// Mitsubishi GX Works2 project: סופי1   PLC: FX3G

// global labels: Global1
VAR_GLOBAL
  LAMP_WORKDAY AT Y007 : BOOL;  (* נורת חווי יום עבודת פעיל *)
  SW_DAY_START AT X007 : BOOL;  (* מתג תחילת יום *)
  SW_START_PROD AT X001 : BOOL;  (* מתג דגימה של Analog Input *)
  SW_EMERGENCY AT X005 : BOOL;  (* מתג חירום לסיום יום עבודה *)
  LAMP_PREP AT Y000 : BOOL;  (* נורת חווי להכנת הגלידה *)
  SW_COOL AT X002 : BOOL;  (* מתג העברת הגלידות למכלי הקירור *)
  TEMP_SENSOR AT X003 : BOOL;  (* חיישן טמפרטורה *)
  LAMP_COOL AT Y002 : BOOL;  (* נורת חווי לקירור גלידה *)
  LAMP_MIX_A AT Y005 : BOOL;  (* נורת הבהוב לערבוב הגלידה *)
  LAMP_MIX_B AT Y006 : BOOL;  (* נורת הבהוב לערבוב הגלידה *)
  INIT_RASBERRY AT D1700 : REAL;  (* רגיסטר מלאי פטל בתחילת יום *)
  INIT_LEMON AT D1702 : REAL;  (* רגיסטר מלאי לימון בתחילת יום *)
  INIT_STABILIZER AT D1705 : REAL;  (* רגיסטר מלאי מייצב בתחילת יום *)
  INIT_BEARS AT D1111 : REAL;  (* רגיסטר מלאי דובונים בתחילת יום *)
  STOCK_RASBERRY AT D1122 : REAL;  (* רגיסטר מלאי נוכחי פטל *)
  STOCK_LEMON AT D1133 : REAL;  (* רגיסטר מלאי נוכחי לימון *)
  STOCK_STABILIZER AT D1233 : REAL;  (* רגיסטר מלאי נוכחי מייצב *)
  STOCK_BEARS AT D1345 : REAL;  (* רגיסטר מלאי נוכחי דובונים *)
  STORAGE_COUNT AT D2000 : REAL;  (* רגיסטר מיכל מארזים *)
  LAMP_REGULAR AT M1 : BOOL;  (* נורת חיווי עזר להכנת גומיגם רגיל *)
  LAMP_PREMIUM AT M2 : BOOL;  (* נורת חיווי להכנת גומיגם פינוק *)
END_VAR
VAR_GLOBAL CONSTANT
  RESET : REAL;  (* איפוס משתנים *)
  RESET_ANALOG_OUTPUT : INT := K0;  (* איפוס משתנים *)
END_VAR
VAR_GLOBAL
  RAS_COOLING_TANK AT D2100 : REAL;  (* מיכל קירור פטל *)
  LEM_COOLING_TANK AT D2200 : REAL;  (* מיכל קירור לימון *)
END_VAR
VAR_GLOBAL CONSTANT
  RAS_FOR_PREMIUIM : REAL := 385;  (* כמות פטל דרושה למארז פינוק *)
  LEM_FOR_PREMIUIM : REAL := 665;  (* כמות לימון דרושה למארז פינוק *)
  STAB_FOR_PREMIUIM : REAL := 210;  (* כמות חומר מייצב להכנת מארז פינוק *)
  RAS_FOR_CLASSIC : REAL := 280;  (* כמות פטל דרושה למארז רגיל *)
  LEM_FOR_CLASSIC : REAL := 455;  (* כמות לימון דרושה מארז רגיל *)
  STAB_FOR_CLASSIC : REAL := 105;  (* כמות חומר מייצב דרושה מארז רגיל *)
END_VAR
VAR_GLOBAL
  ANALOG_INPUT AT D8280 : INT;  (* משתנה המייצג את סוג המארז *)
  ANALOG_OUTPUT AT D8282 : INT;  (* שעון יציאה אנלוגי למספר מארזים *)
  SAVE_ANALOG_INPUT AT D8201 : INT;  (* משתנה שמירת הדגימה שהתקבלה *)
  LACK_OF_STOCK AT M0 : BOOL;  (* נורת חיווי לסיום יום בשל חוסר בחומרי גלם *)
  INDICATOR_LAMP AT M10 : BOOL;  (* נורת חיווי עזר לבדיקת תקינות ערך אנלוגי *)
END_VAR
VAR_GLOBAL CONSTANT
  MAX_REGULAR : REAL := 5;  (* ערך קלט מקסימום ליצירת מארז רגיל *)
  MIN_PREMIUM : REAL := 6;  (* ערך קלט מקסימום ליצירת מארז פינוק *)
END_VAR
VAR_GLOBAL
  ANALOG_SAMPLED AT D8205 : REAL;  (* רגיסטר של המרת ANALOG_INPUT לFLOAT *)
  CHEKING_FOR_REG AT M3 : BOOL;  (* נורת חווי עזר  לבדיקת מלאי להכנת מארז רגיל *)
  CHECKING_FOR_PREM AT M4 : BOOL;  (* נורת חווי לבדיקת מלאי להכנת מארז פינוק *)
  CONTINUE AT M123 : BOOL;  (* נורת חיווי למעבר להפחתת כמויות ממכלים *)
  ITERATION_LIGHT AT M44 : BOOL;  (* נורת חיווי לסיום איטרציה *)
  START_MIX AT M50 : BOOL;  (* נורת חווי עזר להתחלת ערבוב *)
  MAKING_ICECREAM AT M40 : BOOL;  (* נורת חווי להכנת הגלידה *)
END_VAR
VAR_GLOBAL CONSTANT
  TOTAL_REG_LEM : REAL := 490;  (* כמות גלידה לימון במארז רגיל *)
  TOTAL_PREM_LEM : REAL := 700;  (* כמות גלידה לימון במארז פינוק *)
  TOTAL_REG_RAS : REAL := 350;  (* כמות גלידה פטל במארז רגיל *)
  TOTAL_PREM_RAS : REAL := 560;  (* כמות גלידה פטל במארז פינוק *)
  ICECREAM_MAKING_TIME : INT := 50;  (* משך זמן הכנת גלידה *)
END_VAR
VAR_GLOBAL
  SRART_PACKING AT X006 : BOOL;  (* מתג סיום תהליך ואריזה *)
  PACKING_UNIT AT X000 : BOOL;  (* אריזת יחידה *)
  PACKING_LIGHT AT Y001 : BOOL;  (* נורת חווי מסיום אריזת יחידה אחת ועד סיום נורת חווי מאריזת יחידה ועד מארז שלם *)
  COOLING_HELP_LIGHT AT M60 : BOOL;  (* נורת חווי עזר למעבר לקירור *)
  ICECREAM_TIME AT TC1 : BOOL;  (* טיימר שמפעיל את הכנת טעמי הגלידה למשך 5 שניות *)
END_VAR
VAR_GLOBAL CONSTANT
  TOTAL_TIME_ICECREAM : INT := 50;  (* זמן הכנת הגלידות *)
END_VAR
VAR_GLOBAL
  MIXING_DONE AT TS1 : BOOL;  (* הכנת הגלידה הסתיימה *)
  COOLING_DONE AT TS8 : BOOL;  (* זמן הקירור הסתיים *)
  COOLING_TIME AT TC8 : BOOL;  (* טיימר שמפעיל את קירור הגלידות *)
END_VAR
VAR_GLOBAL CONSTANT
  COOLING_TIME_8 : INT := 80;  (* זמן קירור הגלידה *)
END_VAR
VAR_GLOBAL
  MOVE_TO_MIX AT M77 : BOOL;  (* נורת חיווי להעברת הגלידה לערבוב *)
END_VAR
VAR_GLOBAL CONSTANT
  GUMMY_BEAR_FOR_PREMIUM : REAL := 28;  (* כמות דובונים הדרושה למארז רגיל *)
  GUMMY_BEAR_FOR_REGULAR : REAL := 70;  (* כמות דובונים הדרושה למארז פינוק *)
END_VAR
VAR_GLOBAL
  MIXING_FLAVORS AT D1356 : REAL;  (* מיכל ערבוב טעמים *)
  RESET_COOLING AT M88 : BOOL;  (* איפוס מכלי קירור *)
  RAS_ICE_CREAM_STOCK AT D2050 : REAL;  (* מיכל גלידה פטל *)
  LEMON_ICE_CREAM_STOCK AT D2077 : REAL;  (* מיכל גלידה לימון *)
  REG_MIXING_TIME AT TC9 : BOOL;  (* טיימר שמפעיל את ערבוב הגלידות מסוג רגיל *)
  PREM_MIXING_TIME AT TC5 : BOOL;  (* טיימר שמפעיל את ערבוב הגלידות מסוג  פינוק *)
  MIXING_FLAVOUR_DONE1 AT TS9 : BOOL;  (* ערבוב רגיל הסתיים *)
  MIXING_FLAVOUR_DONE2 AT TS5 : BOOL;  (* ערבוב פינוק הסתיים *)
END_VAR
VAR_GLOBAL CONSTANT
  MIX_TIME_3 : INT := 30;  (* זמן ערבוב מארז רגיל *)
  MIX_TIME_5 : INT := 50;  (* זמן ערבוב מארז פינוק *)
END_VAR
VAR_GLOBAL
  FIRST_LIGHT_FLASH AT TC10 : BOOL;  (* הפעלת טיימר הבהוב ראשון *)
  SEC_LIGHT_FLASH AT TC11 : BOOL;  (* הפעלת טיימר הבהוב שני *)
  FIRST_LIGHT_TIMER AT TS10 : BOOL;  (* הבהוב ראשון הסתיים *)
  SEC_LIGHT_TIMER AT TS11 : BOOL;  (* הבהוב שני הסתיים *)
END_VAR
VAR_GLOBAL CONSTANT
  LIGHT_CON : INT := 8;  (* משך זמן הבהוב נורה *)
END_VAR
VAR_GLOBAL
  STORAGE_CONTAINER AT D7777 : REAL;  (* רגיסטר מיכל אחסון *)
END_VAR
VAR_GLOBAL CONSTANT
  PACKAGED_SEVEN_UNIT : REAL := 1;  (* 7 יחידות נארזו *)
  NEW_PAKCAGE : REAL := 1;  (* הוספת מארז מוכן *)
  UNIT_FOR_MESASURE : REAL := 40;  (* קבוע להמרת יחידות מידה *)
END_VAR
VAR_GLOBAL
  UNIT_COUNT AT CC0 : BOOL;  (* ספירת יחידת הגומיגם הראשונה *)
  SEVEN_UNIT_COUNT AT CC1 : BOOL;  (* ספירת 7 יחידות גומיגם *)
  PAC AT CS0 : BOOL;  (* נארזה יחידה *)
  PAC2 AT CS1 : BOOL;  (* נארז מארז *)
  PACK_UNIT AT Y001 : BOOL;  (* נורת חווי מסיום אריזת יחידה אחת ועד סיום נורת חווי מאריזת יחידה ועד מארז שלם *)
END_VAR
VAR_GLOBAL CONSTANT
  RESET_MIXING : REAL;  (* איפוס מיכל *)
  DIVIDER : REAL := 400;  (* מחלק *)
END_VAR
VAR_GLOBAL
  ICECREAMTIME AT TC1 : BOOL;
  FINISH_MIX AT M7 : BOOL;  (* ערבוב נגמר *)
  MIX_LIGHT AT M55 : BOOL;  (* נורת ערבוב *)
END_VAR

// task Task_01 (event TRUE, interval 0, priority 31): POU_01

PROGRAM POU_01
VAR
  StartDay : BOOL;
END_VAR
(* structured ladder/FBD written out as ST: instructions are called as NAME(EN, inputs, outputs); _pN, _eN, _tN stand for wires *)
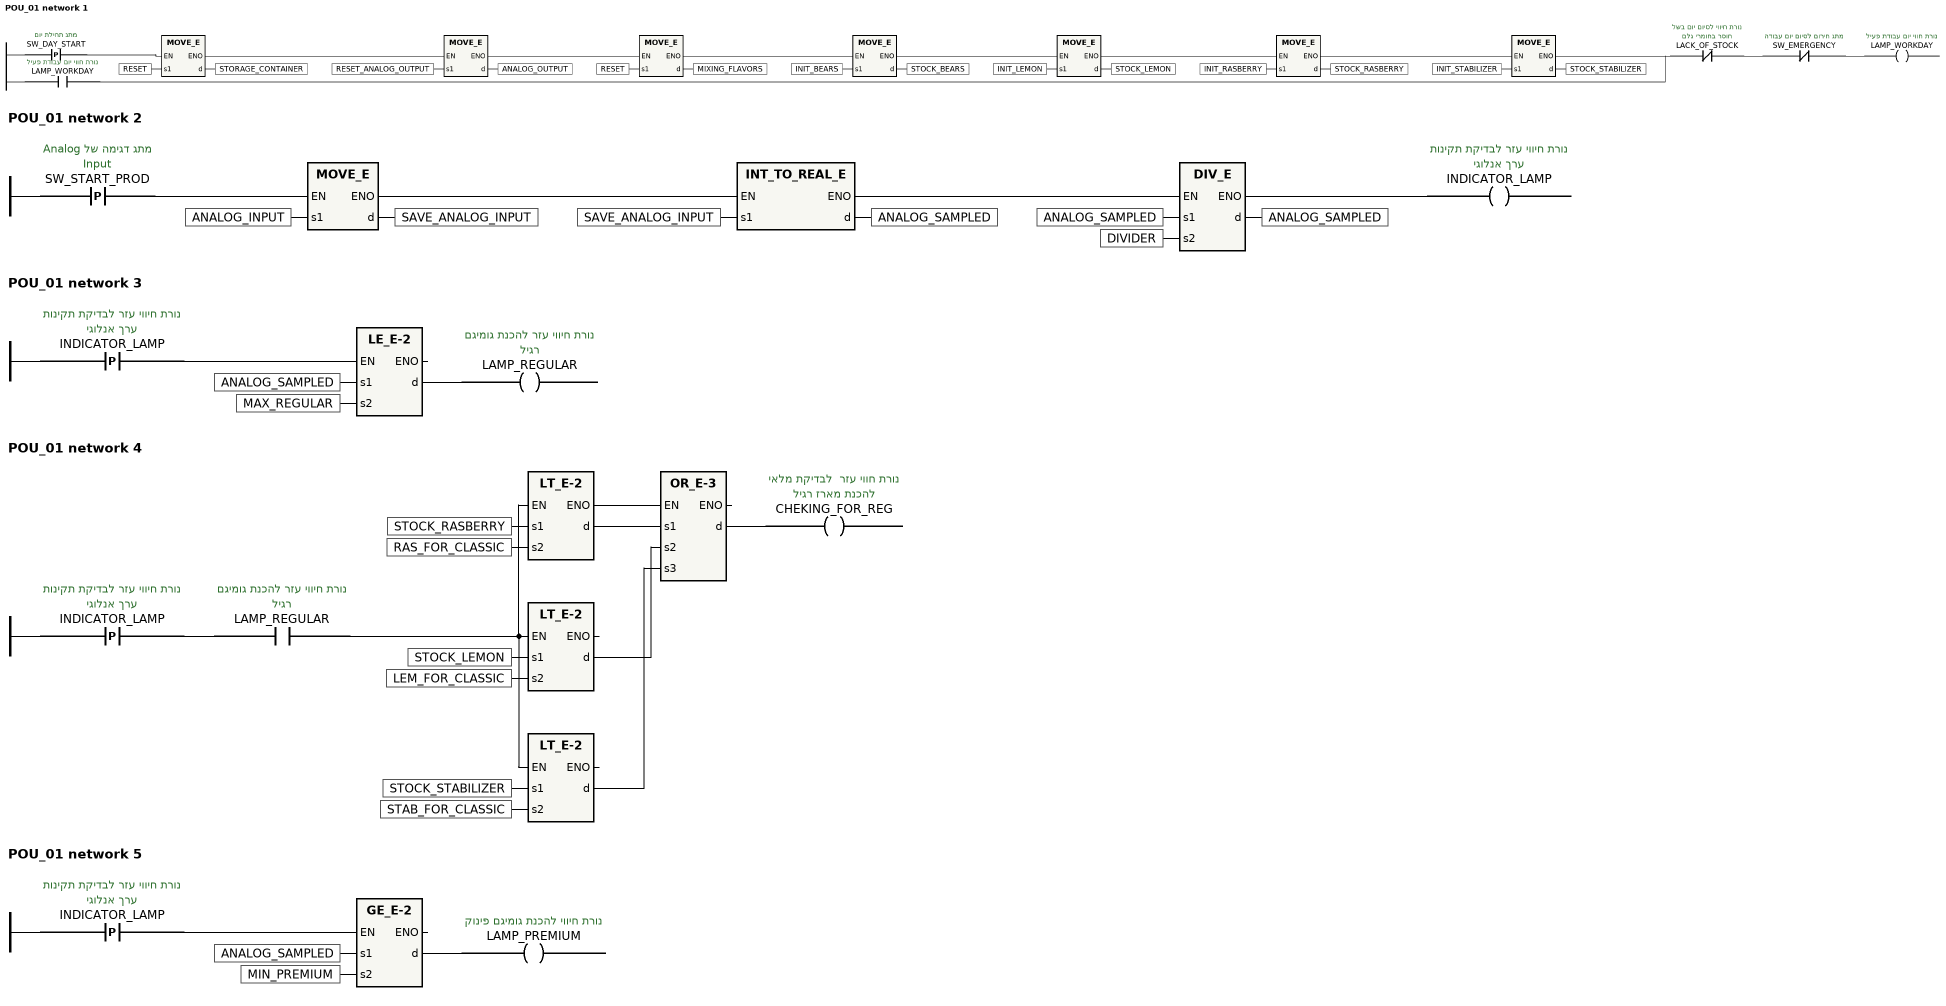
(* network 1 *)
_e1 := MOVE_E(LDP(TRUE, SW_DAY_START), RESET, STORAGE_CONTAINER);
_e2 := MOVE_E(_e1, RESET_ANALOG_OUTPUT, ANALOG_OUTPUT);
_e3 := MOVE_E(_e2, RESET, MIXING_FLAVORS);
_e4 := MOVE_E(_e3, INIT_BEARS, STOCK_BEARS);
_e5 := MOVE_E(_e4, INIT_LEMON, STOCK_LEMON);
_e6 := MOVE_E(_e5, INIT_RASBERRY, STOCK_RASBERRY);
_e7 := MOVE_E(_e6, INIT_STABILIZER, STOCK_STABILIZER);
LAMP_WORKDAY := ((_e7 OR LAMP_WORKDAY) AND NOT LACK_OF_STOCK) AND NOT SW_EMERGENCY;
(* network 2 *)
_e1 := MOVE_E(LDP(TRUE, SW_START_PROD), ANALOG_INPUT, SAVE_ANALOG_INPUT);
_e2 := INT_TO_REAL_E(_e1, SAVE_ANALOG_INPUT, ANALOG_SAMPLED);
_e3 := DIV_E(_e2, ANALOG_SAMPLED, DIVIDER, ANALOG_SAMPLED);
INDICATOR_LAMP := _e3;
(* network 3 *)
LE_E(LDP(TRUE, INDICATOR_LAMP), ANALOG_SAMPLED, MAX_REGULAR, _t1);
LAMP_REGULAR := _t1;
(* network 4 *)
_p1 := LDP(TRUE, INDICATOR_LAMP) AND LAMP_REGULAR;
_e3 := LT_E(_p1, STOCK_RASBERRY, RAS_FOR_CLASSIC, _t2);
LT_E(_p1, STOCK_LEMON, LEM_FOR_CLASSIC, _t4);
LT_E(_p1, STOCK_STABILIZER, STAB_FOR_CLASSIC, _t5);
OR_E(_e3, _t2, _t4, _t5, _t6);
CHEKING_FOR_REG := _t6;
(* network 5 *)
GE_E(LDP(TRUE, INDICATOR_LAMP), ANALOG_SAMPLED, MIN_PREMIUM, _t1);
LAMP_PREMIUM := _t1;
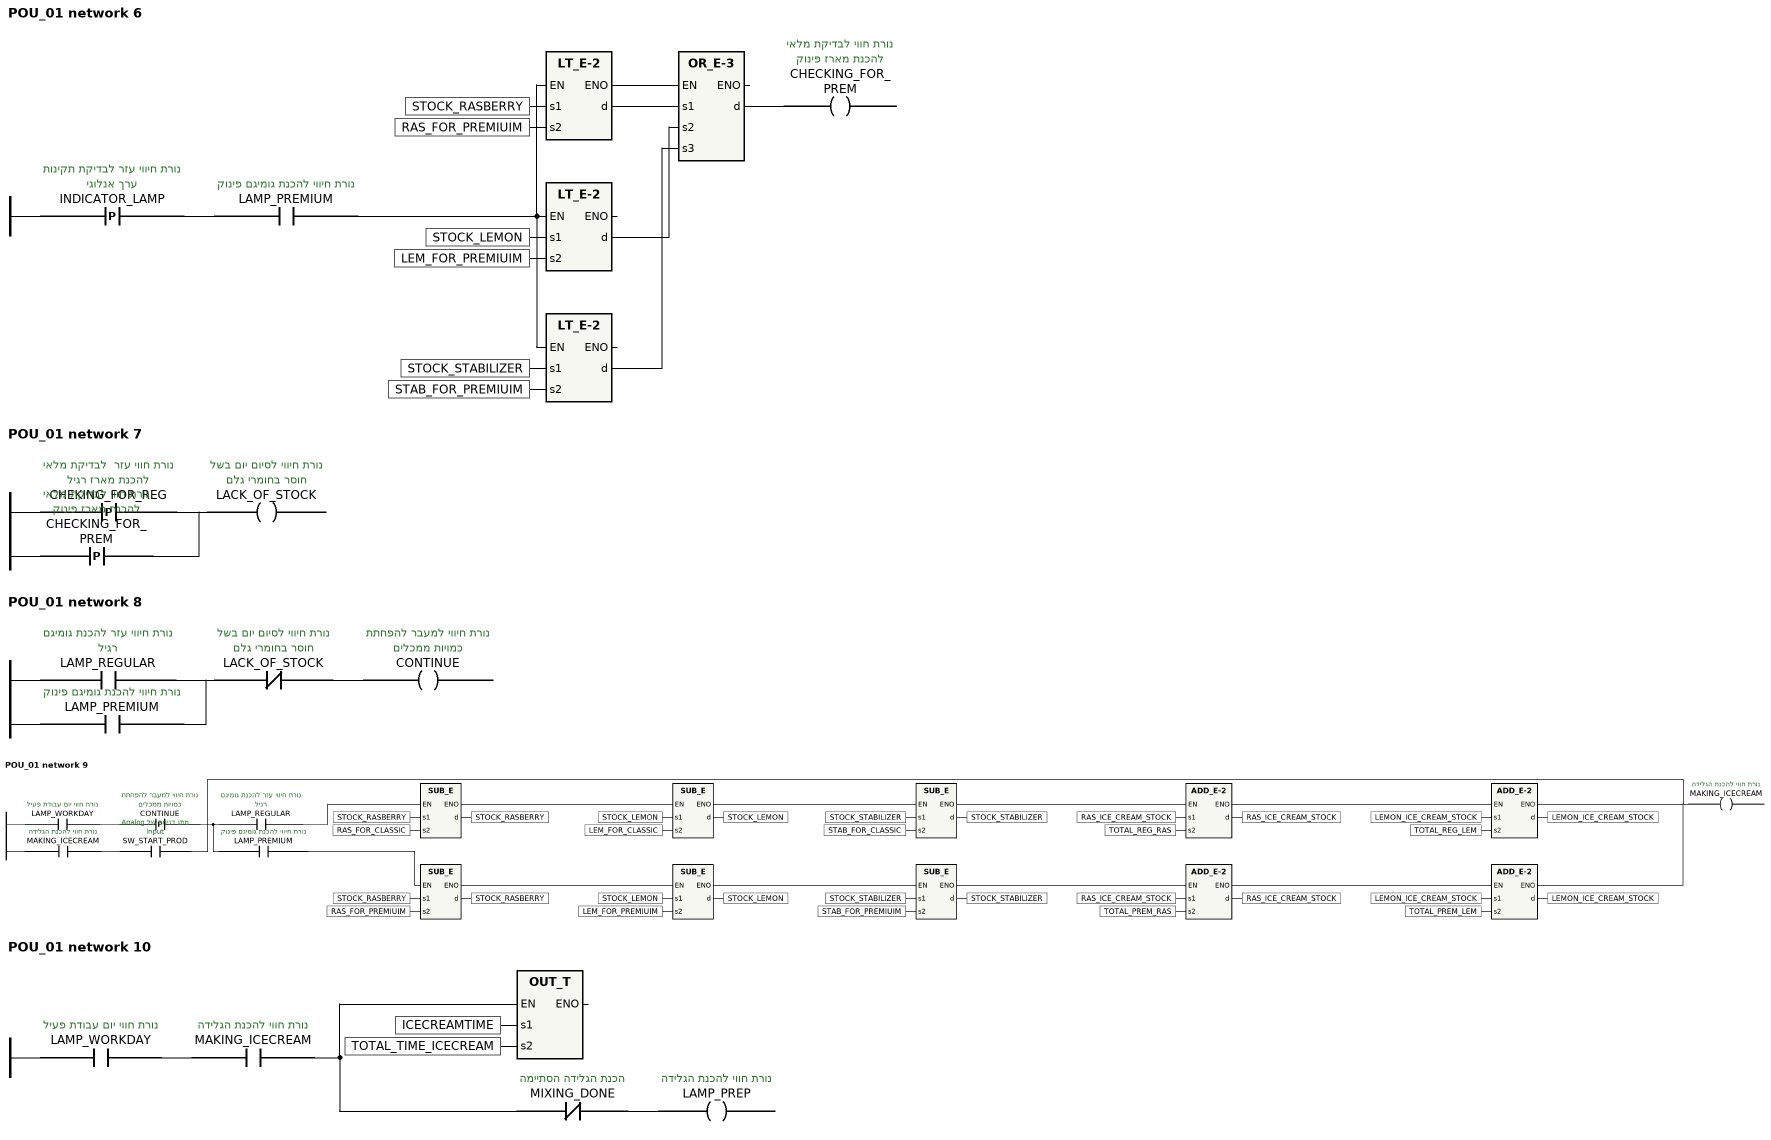
(* network 6 *)
_p1 := LDP(TRUE, INDICATOR_LAMP) AND LAMP_PREMIUM;
_e3 := LT_E(_p1, STOCK_RASBERRY, RAS_FOR_PREMIUIM, _t2);
LT_E(_p1, STOCK_LEMON, LEM_FOR_PREMIUIM, _t4);
LT_E(_p1, STOCK_STABILIZER, STAB_FOR_PREMIUIM, _t5);
OR_E(_e3, _t2, _t4, _t5, _t6);
CHECKING_FOR_PREM := _t6;
(* network 7 *)
LACK_OF_STOCK := LDP(TRUE, CHEKING_FOR_REG) OR LDP(TRUE, CHECKING_FOR_PREM);
(* network 8 *)
CONTINUE := (LAMP_REGULAR OR LAMP_PREMIUM) AND NOT LACK_OF_STOCK;
(* network 9 *)
_p1 := LAMP_WORKDAY AND LDP(TRUE, CONTINUE);
_e2 := SUB_E(_p1 AND LAMP_REGULAR, STOCK_RASBERRY, RAS_FOR_CLASSIC, STOCK_RASBERRY);
_e3 := SUB_E(_e2, STOCK_LEMON, LEM_FOR_CLASSIC, STOCK_LEMON);
_e4 := SUB_E(_e3, STOCK_STABILIZER, STAB_FOR_CLASSIC, STOCK_STABILIZER);
_e5 := ADD_E(_e4, RAS_ICE_CREAM_STOCK, TOTAL_REG_RAS, RAS_ICE_CREAM_STOCK);
_e6 := ADD_E(_e5, LEMON_ICE_CREAM_STOCK, TOTAL_REG_LEM, LEMON_ICE_CREAM_STOCK);
_e7 := SUB_E(_p1 AND LAMP_PREMIUM, STOCK_RASBERRY, RAS_FOR_PREMIUIM, STOCK_RASBERRY);
_e8 := SUB_E(_e7, STOCK_LEMON, LEM_FOR_PREMIUIM, STOCK_LEMON);
_e9 := SUB_E(_e8, STOCK_STABILIZER, STAB_FOR_PREMIUIM, STOCK_STABILIZER);
_e10 := ADD_E(_e9, RAS_ICE_CREAM_STOCK, TOTAL_PREM_RAS, RAS_ICE_CREAM_STOCK);
_e11 := ADD_E(_e10, LEMON_ICE_CREAM_STOCK, TOTAL_PREM_LEM, LEMON_ICE_CREAM_STOCK);
MAKING_ICECREAM := _e6 OR _e11 OR (MAKING_ICECREAM AND SW_START_PROD);
(* network 10 *)
_p1 := LAMP_WORKDAY AND MAKING_ICECREAM;
OUT_T(_p1, ICECREAMTIME, TOTAL_TIME_ICECREAM);
LAMP_PREP := _p1 AND NOT MIXING_DONE;
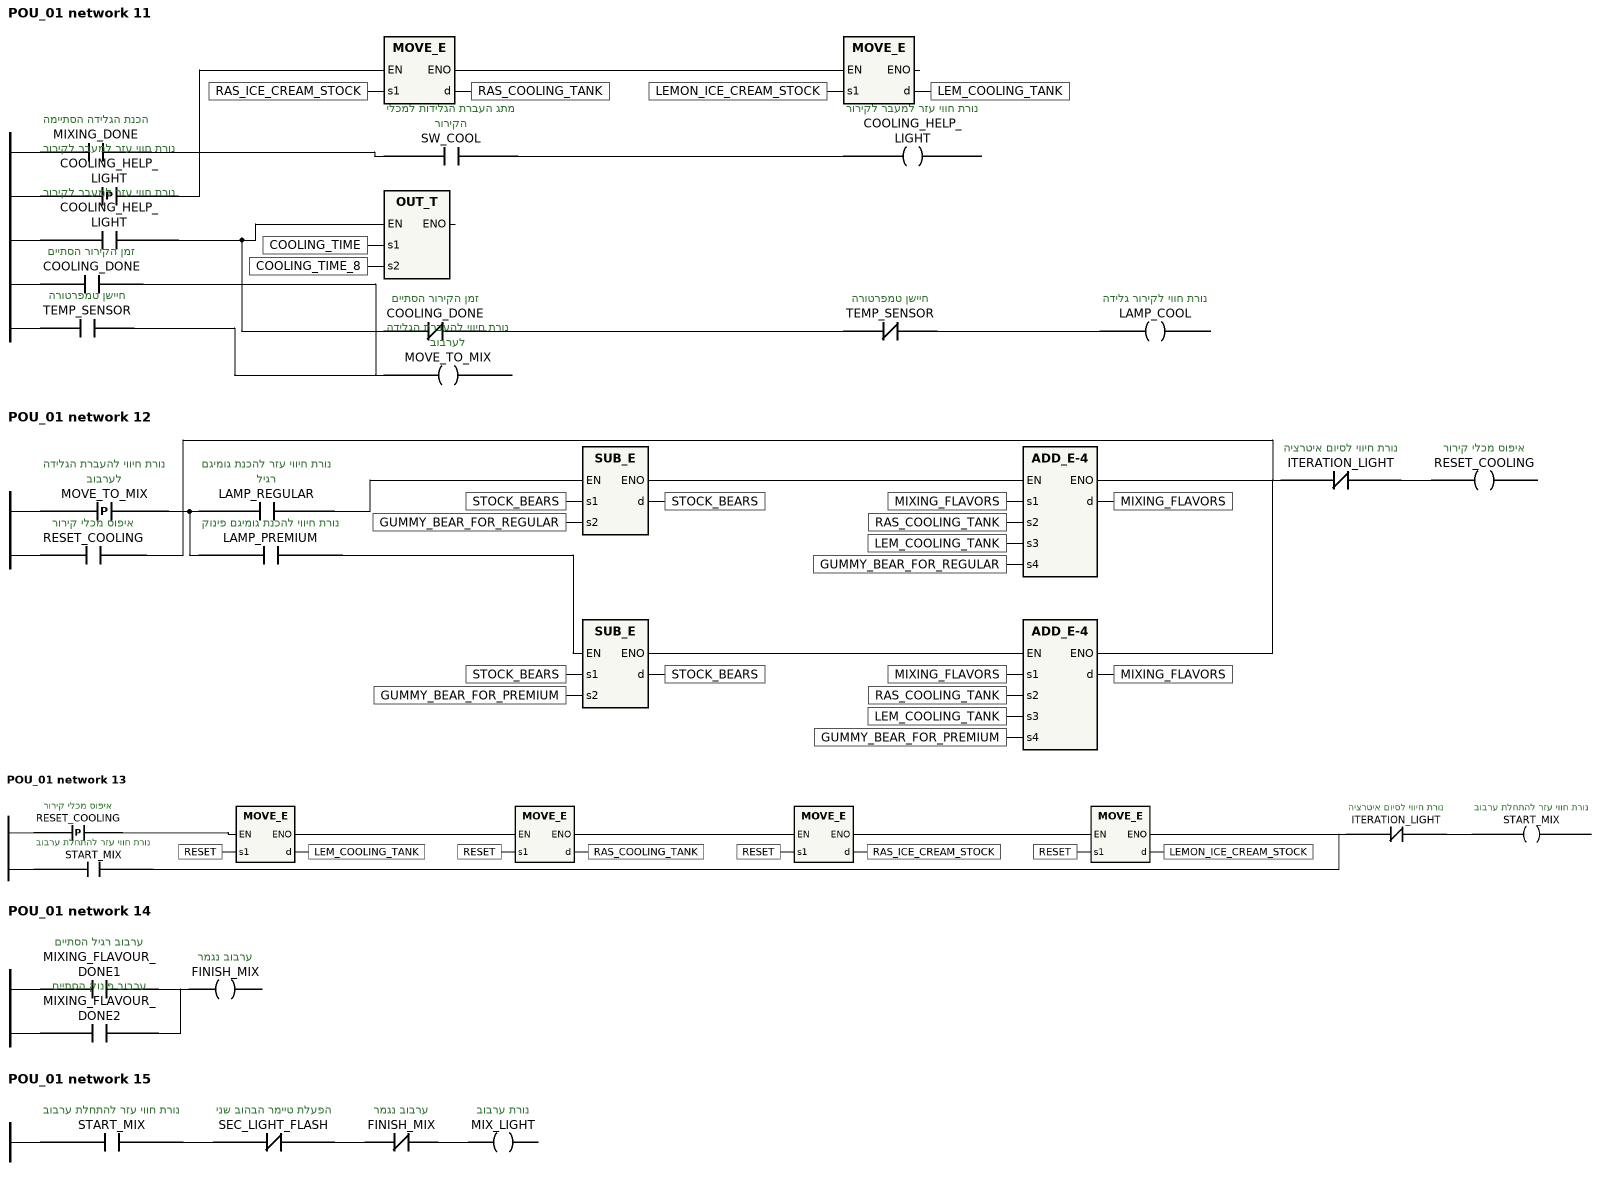
(* network 11 *)
COOLING_HELP_LIGHT := MIXING_DONE AND SW_COOL;
_e1 := MOVE_E(LDP(TRUE, COOLING_HELP_LIGHT), RAS_ICE_CREAM_STOCK, RAS_COOLING_TANK);
MOVE_E(_e1, LEMON_ICE_CREAM_STOCK, LEM_COOLING_TANK);
OUT_T(COOLING_HELP_LIGHT, COOLING_TIME, COOLING_TIME_8);
LAMP_COOL := COOLING_HELP_LIGHT AND NOT COOLING_DONE AND NOT TEMP_SENSOR;
MOVE_TO_MIX := COOLING_DONE OR TEMP_SENSOR;
(* network 12 *)
_p1 := LDP(TRUE, MOVE_TO_MIX);
_e2 := SUB_E(_p1 AND LAMP_REGULAR, STOCK_BEARS, GUMMY_BEAR_FOR_REGULAR, STOCK_BEARS);
_e3 := ADD_E(_e2, MIXING_FLAVORS, RAS_COOLING_TANK, LEM_COOLING_TANK, GUMMY_BEAR_FOR_REGULAR, MIXING_FLAVORS);
_e4 := SUB_E(_p1 AND LAMP_PREMIUM, STOCK_BEARS, GUMMY_BEAR_FOR_PREMIUM, STOCK_BEARS);
_e5 := ADD_E(_e4, MIXING_FLAVORS, RAS_COOLING_TANK, LEM_COOLING_TANK, GUMMY_BEAR_FOR_PREMIUM, MIXING_FLAVORS);
RESET_COOLING := (_e3 OR _e5 OR RESET_COOLING) AND NOT ITERATION_LIGHT;
(* network 13 *)
_e1 := MOVE_E(LDP(TRUE, RESET_COOLING), RESET, LEM_COOLING_TANK);
_e2 := MOVE_E(_e1, RESET, RAS_COOLING_TANK);
_e3 := MOVE_E(_e2, RESET, RAS_ICE_CREAM_STOCK);
_e4 := MOVE_E(_e3, RESET, LEMON_ICE_CREAM_STOCK);
START_MIX := (_e4 OR START_MIX) AND NOT ITERATION_LIGHT;
(* network 14 *)
FINISH_MIX := MIXING_FLAVOUR_DONE1 OR MIXING_FLAVOUR_DONE2;
(* network 15 *)
MIX_LIGHT := START_MIX AND NOT SEC_LIGHT_FLASH AND NOT FINISH_MIX;
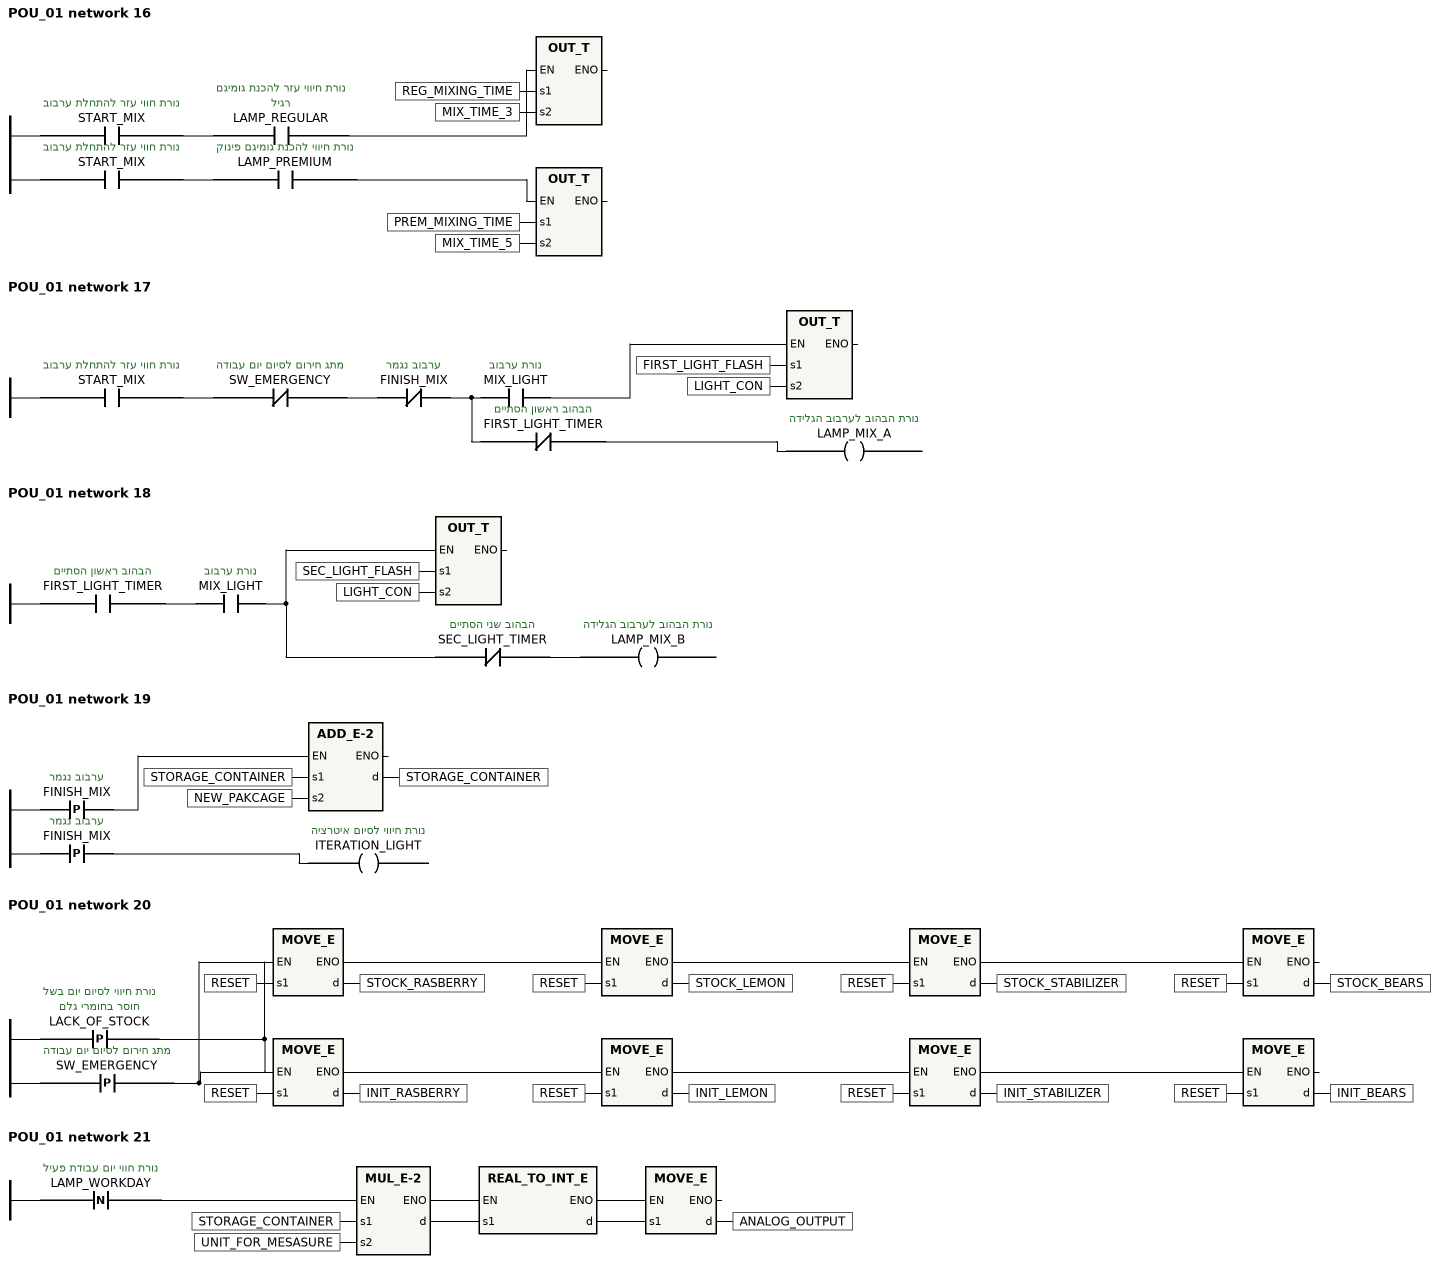
(* network 16 *)
OUT_T(START_MIX AND LAMP_REGULAR, REG_MIXING_TIME, MIX_TIME_3);
OUT_T(START_MIX AND LAMP_PREMIUM, PREM_MIXING_TIME, MIX_TIME_5);
(* network 17 *)
_p1 := START_MIX AND NOT SW_EMERGENCY AND NOT FINISH_MIX;
OUT_T(_p1 AND MIX_LIGHT, FIRST_LIGHT_FLASH, LIGHT_CON);
LAMP_MIX_A := _p1 AND NOT FIRST_LIGHT_TIMER;
(* network 18 *)
_p1 := FIRST_LIGHT_TIMER AND MIX_LIGHT;
OUT_T(_p1, SEC_LIGHT_FLASH, LIGHT_CON);
LAMP_MIX_B := _p1 AND NOT SEC_LIGHT_TIMER;
(* network 19 *)
ADD_E(LDP(TRUE, FINISH_MIX), STORAGE_CONTAINER, NEW_PAKCAGE, STORAGE_CONTAINER);
ITERATION_LIGHT := LDP(TRUE, FINISH_MIX);
(* network 20 *)
_p1 := LDP(TRUE, LACK_OF_STOCK) OR LDP(TRUE, SW_EMERGENCY);
_e2 := MOVE_E(_p1, RESET, STOCK_RASBERRY);
_e3 := MOVE_E(_e2, RESET, STOCK_LEMON);
_e4 := MOVE_E(_e3, RESET, STOCK_STABILIZER);
MOVE_E(_e4, RESET, STOCK_BEARS);
_e5 := MOVE_E(_p1, RESET, INIT_RASBERRY);
_e6 := MOVE_E(_e5, RESET, INIT_LEMON);
_e7 := MOVE_E(_e6, RESET, INIT_STABILIZER);
MOVE_E(_e7, RESET, INIT_BEARS);
(* network 21 *)
_e2 := MUL_E(LDF(TRUE, LAMP_WORKDAY), STORAGE_CONTAINER, UNIT_FOR_MESASURE, _t1);
_e4 := REAL_TO_INT_E(_e2, _t1, _t3);
MOVE_E(_e4, _t3, ANALOG_OUTPUT);
END_PROGRAM
